TEXTLIST AccessPanelCmbTxtList
  1 = '1'
  2 = '2'
  3 = '3'
  4 = '4'
   = ''
END_TEXTLIST

(* stored: Version 1.1.0.1, ProductVersion 3.1.4024.4
   TextList AccessPanelCmbTxtList: Id {87e19387-2f05-434e-a3af-f07ed2b71d17} *)
